// TIA Portal V20 export
VAR_GLOBAL   // PLC tag table "LExample_Constants"
END_VAR
VAR_GLOBAL CONSTANT   // user constants
   MAX_LExample : DInt := 4;   // Constant LExample
END_VAR
